SUBAPPLICATION mapping_Uebung_029 (* LED_DO Blinkende LED *)
  (* Standard: 61499-2; Description: Copyright (c) 2023 Meisterschulen am Ostbahnhof This program and the accompanying materials are made available under the terms of the Eclipse Public License 2.0 which is available at https://www.eclipse.org/legal/epl-2.0/ SPDX-License-Identifier: EPL-2.0 *)
  (* Version 1.0, 2023-10-23, Franz Höpfinger, Meisterschulen am Ostbahnhof *)
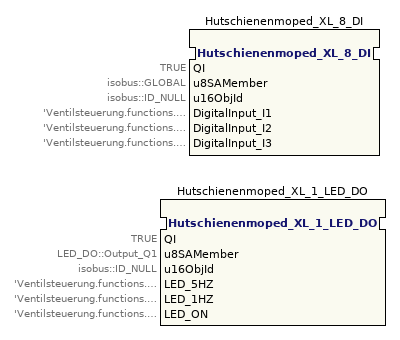
  FBS
    Hutschienenmoped_XL_8_DI : Hutschienenmoped_XL_8_DI(QI := TRUE, u8SAMember := isobus::GLOBAL, u16ObjId := isobus::ID_NULL, DigitalInput_I1 := 'Ventilsteuerung.functions.DigitalInput_I1', DigitalInput_I2 := 'Ventilsteuerung.functions.DigitalInput_I2', DigitalInput_I3 := 'Ventilsteuerung.functions.DigitalInput_I3');
    Hutschienenmoped_XL_1_LED_DO : Hutschienenmoped_XL_1_LED_DO(QI := TRUE, u8SAMember := LED_DO::Output_Q1, u16ObjId := isobus::ID_NULL, LED_5HZ := 'Ventilsteuerung.functions.LED_Q1_5HZ', LED_1HZ := 'Ventilsteuerung.functions.LED_Q1_1HZ', LED_ON := 'Ventilsteuerung.functions.LED_Q1_ON');
  END_FBS
END_SUBAPPLICATION
